// TIA Portal V18 export
TYPE "Check"
// stored: IsFailsafeCompliant false
   STRUCT
      Mode : Bool;   // 防错模式
      DataClear : Bool;   // 数据清除
      Code : Array[0..10] of String[48];   // 防错码
      Choice1 : Bool;   // 防错项选择
      Choice2 : Bool;
      Choice3 : Bool;
      Choice4 : Bool;
      Choice5 : Bool;
      Choice6 : Bool;
      Choice7 : Bool;
      Choice8 : Bool;
      TotalResult : Array[0..10] of Int;   // 防错项结果
      OP2Result : Array[0..10] of Int;
      OP5Result : Array[0..10] of Int;
      AllResult : Int;   // 防错项总结果
      LoadInx : Int;
   END_STRUCT;
END_TYPE
